FUNCTION_BLOCK Manager
  (* Standard: 61499-2 *)
  (* Version 0.1, 2017-00-02, hpea485, UOA *)
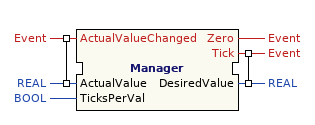
  EVENT_INPUT
    ActualValueChanged WITH ActualValue;
  END_EVENT
  EVENT_OUTPUT
    Zero;
    Tick WITH DesiredValue;
  END_EVENT
  VAR_INPUT
    ActualValue : REAL;
    TicksPerVal : BOOL := 100;
  END_VAR
  VAR_OUTPUT
    DesiredValue : REAL;
  END_VAR
  VAR
    Len : INT := 10;
    Pos : INT := 0;
    Vals : ARRAY [0..9] OF REAL := [1.0,2.5,3.0,4.0,-5.0,-1.0,3.0,8.0,9.0,-5.5];
    TickCount : INT;
  END_VAR
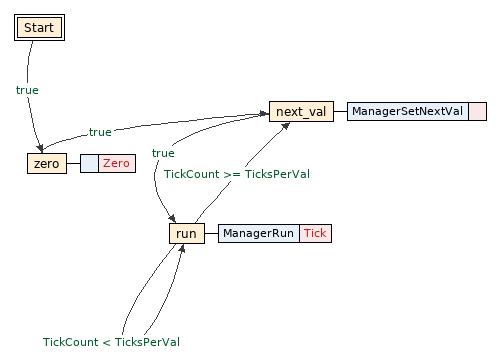
  EC_STATES
    Start;
    next_val : ManagerSetNextVal;
    run : ManagerRun -> Tick;
    zero : -> Zero;
  END_STATES
  EC_TRANSITIONS
    Start TO zero := true;
    next_val TO run := true;
    run TO next_val := TickCount >= TicksPerVal;
    run TO run := TickCount < TicksPerVal;
    zero TO next_val := true;
  END_TRANSITIONS
  ALGORITHM ManagerSetNextVal IN C:
me->DesiredValue = me->Vals[me->Pos];
me->Pos++;
if(me->Pos >= me->Len) {
	me->Pos = 0;
}
me->TickCount = 0;
printf("NEW DESIRE\nSetting Desired Value to %f\n", me->DesiredValue);
  END_ALGORITHM
  ALGORITHM ManagerRun IN C:
printf("Tick:\t%i\tDesired:\t%f\tActual:\t%f\n", me->TickCount, me->DesiredValue, me->ActualValue);
me->TickCount++;
  END_ALGORITHM
END_FUNCTION_BLOCK
